Staubli VAL3: loadmaster8.pgx

program loadmaster8(string x_sMasterFile8 (dimensions=1))
begin
  if master:libLoad(x_sMasterFile8)<0
    popUpMsg("nO ok")
  endIf
  frmaster[8].trsf=master:tTool.trsf
  //取个数
  nsize[8]=size(master:ptRoutingPath)
  //存个数
  resize(pdemo8,1,nsize[8])
  //保存程序
  master:libSave()
end
